FUNCTION S_POSITION3D_TO_S_POSITION2D : S_POSITION2D
VAR_INPUT
	IN_VALUE : S_POSITION2D;
END_VAR
VAR
END_VAR

S_POSITION3D_TO_S_POSITION2D := IN_VALUE;

END_FUNCTION

(* stored: Version 1.1.0.1, ProductVersion 3.1.4019.2
   POU S_POSITION3D_TO_S_POSITION2D: Id {deef4e32-65bb-40eb-9440-3da9ea46c4c4}, SpecialFunc None *)
